# B&R Automation Studio project laba 1
Automation Studio 4.5.2.102

## Configuration Config1

### Task classes (Cpu.sw)
```
Cyclic#1:
  Program <- Program.prg
Binaries: udbdef, TCData, ashwd, User, asfw, arconfig, sysconf, Role, ashwac, iomap
Libraries: Library
```

### Hardware
```
4PP065_0571_P74 : 4PP065.0571-P74 v1.1.2.0
  Connector IF5:
    ActivateDevice = 1
  ConfigurationID = labBR
  Simulation = 1
```

## Logical view

### Library Logical/Libraries/Library

#### Library.fun
```iecst
{REDUND_ERROR} {REDUND_UNREPLICABLE} FUNCTION_BLOCK FB_Integrator (*TODO: Add your comment here*) (*$GROUP=User,$CAT=User,$GROUPICON=User.png,$CATICON=User.png*)
	VAR_INPUT
		in : {REDUND_UNREPLICABLE} REAL;
	END_VAR
	VAR_OUTPUT
		out : {REDUND_UNREPLICABLE} REAL;
	END_VAR
	VAR
		dt : {REDUND_UNREPLICABLE} REAL;
	END_VAR
END_FUNCTION_BLOCK

{REDUND_ERROR} {REDUND_UNREPLICABLE} FUNCTION_BLOCK FB_Motor (*TODO: Add your comment here*) (*$GROUP=User,$CAT=User,$GROUPICON=User.png,$CATICON=User.png*)
	VAR_INPUT
		u : {REDUND_UNREPLICABLE} REAL;
	END_VAR
	VAR_OUTPUT
		w : {REDUND_UNREPLICABLE} REAL;
		phi : {REDUND_UNREPLICABLE} REAL;
	END_VAR
	VAR
		integrator : {REDUND_UNREPLICABLE} FB_Integrator;
		Tm : {REDUND_UNREPLICABLE} REAL;
		ke : {REDUND_UNREPLICABLE} REAL;
		dt : {REDUND_UNREPLICABLE} REAL;
	END_VAR
END_FUNCTION_BLOCK

{REDUND_ERROR} {REDUND_UNREPLICABLE} FUNCTION_BLOCK FB_Regulator (*TODO: Add your comment here*) (*$GROUP=User,$CAT=User,$GROUPICON=User.png,$CATICON=User.png*)
	VAR_INPUT
		e : {REDUND_UNREPLICABLE} REAL;
	END_VAR
	VAR_OUTPUT
		u : {REDUND_UNREPLICABLE} REAL;
	END_VAR
	VAR
		k_i : {REDUND_UNREPLICABLE} REAL;
		integrator : {REDUND_UNREPLICABLE} FB_Integrator;
		iyOld : {REDUND_UNREPLICABLE} REAL;
		max_abs_value : {REDUND_UNREPLICABLE} REAL;
		dt : {REDUND_UNREPLICABLE} REAL;
		k_p : {REDUND_UNREPLICABLE} REAL;
	END_VAR
END_FUNCTION_BLOCK
```

#### FB_Integrator.c
```c
#include <bur/plctypes.h>
#ifdef __cplusplus
	extern "C"
	{
#endif
	#include "Library.h"
#ifdef __cplusplus
	};
#endif
/* TODO: Add your comment here */
void FB_Integrator(struct FB_Integrator* inst)
{
	/*TODO: Add your code here*/
	inst->out = inst->dt * inst->in + inst->out;
}
```

#### FB_Motor.c
```c
#include <bur/plctypes.h>
#ifdef __cplusplus
	extern "C"
	{
#endif
	#include "Library.h"
#ifdef __cplusplus
	};
#endif
/* TODO: Add your comment here */
void FB_Motor(struct FB_Motor* inst)
{
	/*TODO: Add your code here*/
	REAL A = (inst->u / inst->ke - inst->w) / inst->Tm;
	inst->integrator.in = A;
	FB_Integrator(&inst->integrator);

	inst->w = inst->integrator.out;
}
```

#### FB_Regulator.c
```c
#include <bur/plctypes.h>
#ifdef __cplusplus
	extern "C"
	{
#endif
	#include "Library.h"
#ifdef __cplusplus
	};
#endif
/* TODO: Add your comment here */

REAL LimitValue(REAL max, REAL x)
{
	if (x > max)
	{
		x = max;
	}
	if (x < -max)
	{
		x = -max;
	}
	return x;
}

void FB_Regulator(struct FB_Regulator* inst)
{
	/*TODO: Add your code here*/
	REAL A = inst->e * inst->k_p;
	REAL B = inst->e * inst->k_i;

	A = LimitValue(inst->max_abs_value, A);

	inst->integrator.in = B + inst->iyOld;
	FB_Integrator(&inst->integrator);

	A = A + inst->integrator.out;

	inst->u = LimitValue(inst->max_abs_value, A);

	inst->iyOld = inst->u - A;

}
```

### Program Logical/Program

#### Variables.var
```iecst
VAR
	fb_controller : FB_Regulator;
	fb_motor1 : FB_Motor;
	Speed : REAL;
	Enable : BOOL;
	counter : UINT;
	fb_motor2 : FB_Motor;
END_VAR
```

#### Cyclic.c
```c
#include <bur/plctypes.h>

#ifdef _DEFAULT_INCLUDES
	#include <AsDefault.h>
#endif

void _CYCLIC ProgramCyclic(void)
{
	if(Enable)
	{
		if  (counter == 400)
		{
			Speed = 0;
			counter = 0;
		}
		if (counter == 200)
		{
			Speed = 40;
		}

		fb_motor1.u = Speed * fb_motor1.ke;
		FB_Motor(& fb_motor1);

		fb_controller.e = Speed - fb_motor2.w;
		FB_Regulator(& fb_controller);
		fb_motor2.u = fb_controller.u;
		FB_Motor(& fb_motor2);

		counter ++;

	}
}
```

#### Init.c
```c
#include <bur/plctypes.h>

#ifdef _DEFAULT_INCLUDES
	#include <AsDefault.h>
#endif

void _INIT ProgramInit(void)
{
	fb_motor1.dt = 0.01;
	fb_motor1.ke = 0.24;
	fb_motor1.Tm = 0.1;
	fb_motor1.u = 0;
	fb_motor1.integrator.dt=0.01;

	fb_motor2.dt = 0.01;
	fb_motor2.ke = 0.24;
	fb_motor2.Tm = 0.1;
	fb_motor2.u = 0;
	fb_motor2.integrator.dt=0.01;

	fb_controller.dt = 0.01;
	fb_controller.integrator.dt = 0.01;
	fb_controller.k_i = 2.7;
	fb_controller.k_p = 0.3;
	fb_controller.max_abs_value = 24.0;

	Speed = 0;
	counter = 0;
	Enable = 1;
}
```
